FUNCTION_BLOCK Controller
  (* Standard: 61499-2 *)
  (* Version 0.1, 2015-00-14, Th?o, PC_THEO *)
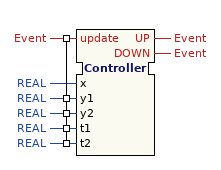
  EVENT_INPUT
    update WITH y1, y2, t1, t2;
  END_EVENT
  EVENT_OUTPUT
    UP;
    DOWN;
  END_EVENT
  VAR_INPUT
    x : REAL;
    y1 : REAL;
    y2 : REAL;
    t1 : REAL;
    t2 : REAL;
  END_VAR
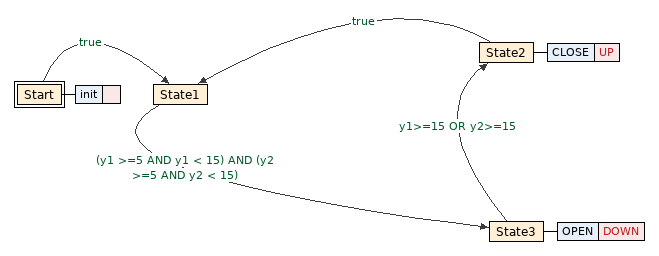
  EC_STATES
    Start : init;
    State1;
    State2 : CLOSE -> UP;
    State3 : OPEN -> DOWN;
  END_STATES
  EC_TRANSITIONS
    Start TO State1 := true;
    State1 TO State3 := (y1 >=5 AND y1 < 15) AND (y2 >=5 AND y2 < 15);
    State2 TO State1 := true;
    State3 TO State2 := y1>=15 OR y2>=15;
  END_TRANSITIONS
  ALGORITHM init IN C:
me->y1=0;
me->y2=0;
  END_ALGORITHM
  ALGORITHM OPEN IN C:
if(me->t1>me->t2){
printf("signal sent : open the gate, y1 : %f, y2 : %f, time : %f\n", me->y1, me->y2, me->t1);
}else{
printf("signal sent : open the gate, y1 : %f, y2 : %f, time : %f\n", me->y1, me->y2, me->t2);
}
  END_ALGORITHM
  ALGORITHM CLOSE IN C:
if(me->t1>me->t2){
printf("signal sent : close the gate, y1 : %f, y2 : %f, time : %f\n", me->y1, me->y2, me->t1);
}else{
printf("signal sent : close the gate, y1 : %f, y2 : %f, time : %f\n", me->y1, me->y2, me->t2);
}
  END_ALGORITHM
END_FUNCTION_BLOCK
